Fanuc KAREL source: kt00376.KL

-- PROVISIONAL review KL for V770-1; original PC SHA256 76c6efb2cecc90a095339375651aacb885ab3652f2a6e20ee53351566435706d
-- Incomplete behavior may be omitted. Consult companion uncertainty JSON. Do not deploy.
PROGRAM KT00376
%NOLOCKGROUP
VAR
  R2 : REAL
  OUT : BOOLEAN
-- UNRESOLVED_DECL Y1 type=002018
BEGIN
  -- UNRESOLVED_PC offsets 5-19; opcodes 2E,22,9D,33,B2
  -- UNRESOLVED_PC offsets 24-35; opcodes 2E,23
  -- UNRESOLVED_PC offsets 40-65; opcodes 22,9D,33,B1,21,29,64,29,70,23
  -- UNRESOLVED_PC offsets 70-74; opcodes 7F
END KT00376
